// TIA Portal V17 export
// export: Created 2026-04-13T11:12:41.3675698Z, ExportSetting WithDefaults, DisplayName Totally Integrated Automation Portal, DisplayVersion V17 Update 4, DisplayName TIA Portal Openness, DisplayVersion V17 Update 4, DisplayName TIA Portal Version Control Interface, DisplayVersion V17, DisplayName SINAMICS Startdrive Advanced, DisplayVersion V17, DisplayName SINAMICS Startdrive G130, G150, S120, S150, SINAMICS MV, S210, DisplayVersion V17, DisplayName SINAMICS Startdrive G110M, G120, G120C, G120D, G120P, G115D, DisplayVersion V17, DisplayName STEP 7 Professional, DisplayVersion V17 Update 4, DisplayName STEP 7 Safety, DisplayVersion V17, DisplayName WinCC Professional, DisplayVersion V17 Update 4
FUNCTION_BLOCK "A2-数据转换RTI"   // FB48, SCL
{ S7_Optimized_Access := 'TRUE' }
VERSION : 0.1
// stored: AutoNumber true, IsIECCheckEnabled false, IsRetainMemResEnabled false, MemoryReserve 100, SetENOAutomatically false, UDAEnableTagReadback false
   VAR_INPUT
      I_Max : Int := 27648;
      I_Min : Int := 0;
      R_Max : Real;
      R_Min : Real;
      R_Value : Real;
   END_VAR
   VAR_OUTPUT
      I_ChValue : Int;
   END_VAR
BEGIN
   (**)
   #I_ChValue := REAL_TO_INT((#R_Value - #R_Min) / (#R_Max - #R_Min) *( #I_Max-#I_Min))+#I_Min;
   (* OUT = [((FLOAT (IN) – K1)/(K2–K1)) * (HI_LIM–LO_LIM)] + LO_LIM *)
END_FUNCTION_BLOCK
